FUNCTION_BLOCK PUBLIC set_qr_info

VAR
	modified_qr:DINT;
	
END_VAR

   IF(pf_x_angle_valid=1 AND pf_y_tag_valid=1) THEN 
	lastqrtagtime := F_GetSystemTime() ;
 // END_IF	
 // IF(raw_qr_tag<>0 AND ((robotdata.robot_direction MOD 2 =0 AND robotdata.qr_x<>0) OR (robotdata.robot_direction MOD 2 =1 AND robotdata.qr_y<>0))) THEN
  	modified_qr:=raw_qr_tag;
    IF(raw_qr_tag>=82 AND raw_qr_tag<102)  THEN
      robotdata.qr_tag := raw_qr_tag-61;
      grid_x := (robotdata.qr_tag-1)/5;
      grid_y := (robotdata.qr_tag-1) MOD 5;
    
    ELSIF(raw_qr_tag>101)THEN
      modified_qr := raw_qr_tag-102;
      robotdata.qr_tag := raw_qr_tag-61;
      grid_x := (modified_qr)/4;
      grid_y := (modified_qr) MOD 4+5;
    ELSIF(raw_qr_tag>40)THEN
      grid_x := (robotdata.qr_tag-41)/4;
      grid_y := (robotdata.qr_tag-41) MOD 4+5;
     robotdata.qr_tag :=raw_qr_tag;
    ELSE
	grid_x := (robotdata.qr_tag-1)/5;
    grid_y := (robotdata.qr_tag-1) MOD 5;
	robotdata.qr_tag :=raw_qr_tag;
	END_IF
    robotdata.qr_yaw :=  LMOD((-robotdata.qr_angle * 0.1-PF_OFFSET) * PI / 180.0+(2*PI) , (2*PI));
    robotdata.robot_x := (grid_x * GRID_DIM) + (robotdata.qr_x / 1000.0) + (robotdata.encoder_v * COS(robotdata.qr_yaw) * PLC_CYCLE ); //the constant at the end is based on the latency of the camera
    robotdata.robot_yaw:=robotdata.qr_yaw;
    IF(  NOT winnerEvaluated AND ABS(robotdata.imux_rel-(robotdata.qr_x / 1000.0))<ABS(robotdata.encoderx_rel-(robotdata.qr_x / 1000.0))) THEN
      imuXwins:=TRUE;
    ELSIF( NOT winnerEvaluated AND ABS(robotdata.imux_rel-(robotdata.qr_x / 1000.0))>ABS(robotdata.encoderx_rel-(robotdata.qr_x / 1000.0))) THEN
      imuXwins:=FALSE;
	  END_IF
    
    robotdata.encoder_x := robotdata.robot_x;
    robotdata.imu_state.imu_x := robotdata.robot_x;
	
  
  
    robotdata.robot_y := (grid_y * GRID_DIM) + (robotdata.qr_y / 1000.0) + (robotdata.encoder_v * SIN(robotdata.qr_yaw) * PLC_CYCLE);
    IF( NOT winnerEvaluated AND  ABS(robotdata.imuy_rel-(robotdata.qr_y / 1000.0))<ABS(robotdata.encodery_rel-(robotdata.qr_y / 1000.0))) THEN
      imuYwins:=TRUE;
    ELSIF( NOT winnerEvaluated AND  ABS(robotdata.imuy_rel-(robotdata.qr_y / 1000.0))>ABS(robotdata.encodery_rel-(robotdata.qr_y / 1000.0))) THEN
      imuYwins:=FALSE;
	END_IF   
  
    winnerEvaluated:=TRUE;

   //printf("%d-%d\n",imuXwins,imuYwins);
    robotdata.encoder_y := robotdata.robot_y;
    robotdata.imu_state.imu_y :=robotdata.robot_y;
	//robotdata.imu_state.imu_euler:=robotdata.robot_yaw;
	robotdata.encoder_yaw:=robotdata.robot_yaw;
	//robotdata.encoder_yaw:=robotdata.qr_yaw;
    //imu_odometry->imu_euler=qr_info->yaw_state;
   ELSE
    winnerEvaluated:=FALSE;
	robotdata.qr_tag :=0;
	END_IF

END_FUNCTION_BLOCK

(* stored: Version 1.1.0.1, ProductVersion 3.1.4024.12
   POU set_qr_info: Id {2c1e8f8b-2e44-47c9-b13d-0d890683b045}, SpecialFunc None *)
